FUNCTION_BLOCK MM_TO_PLS
VAR_INPUT
	UINT_PLS_RATIO : UINT;
	UINT_TARGET1_MM : UINT;
	UINT_VEL1_MM : UINT;
	UINT_TARGET2_MM : UINT;
	UINT_VEL2_MM : UINT;
	UINT_TARGET3_MM : UINT;
	UINT_VEL3_MM : UINT;
	UINT_TARGET4_MM : UINT;
	UINT_VEL4_MM : UINT;
	UINT_JOG_2SPD_MM : UINT;
END_VAR

VAR_OUTPUT
	TARGET1_WR_UINT : UINT;
	VEL1_WR_UINT : UINT;
	TARGET2_WR_UINT : UINT;
	VEL2_WR_UINT : UINT;
	TARGET3_WR_UINT : UINT;
	VEL3_WR_UINT : UINT;
	TARGET4_WR_UINT : UINT;
	VEL4_WR_UINT : UINT;
	JOG_2SPD_UINT : UINT;

END_VAR

VAR
END_VAR

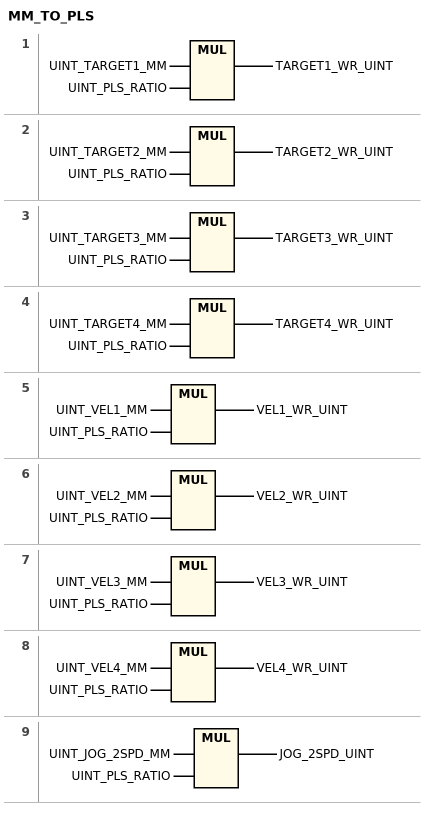
// NETWORK 1
TARGET1_WR_UINT := UINT_TARGET1_MM * UINT_PLS_RATIO;

// NETWORK 2
TARGET2_WR_UINT := UINT_TARGET2_MM * UINT_PLS_RATIO;

// NETWORK 3
TARGET3_WR_UINT := UINT_TARGET3_MM * UINT_PLS_RATIO;

// NETWORK 4
TARGET4_WR_UINT := UINT_TARGET4_MM * UINT_PLS_RATIO;

// NETWORK 5
VEL1_WR_UINT := UINT_VEL1_MM * UINT_PLS_RATIO;

// NETWORK 6
VEL2_WR_UINT := UINT_VEL2_MM * UINT_PLS_RATIO;

// NETWORK 7
VEL3_WR_UINT := UINT_VEL3_MM * UINT_PLS_RATIO;

// NETWORK 8
VEL4_WR_UINT := UINT_VEL4_MM * UINT_PLS_RATIO;

// NETWORK 9
JOG_2SPD_UINT := UINT_JOG_2SPD_MM * UINT_PLS_RATIO;

END_FUNCTION_BLOCK

(* stored: Version 1.1.0.1, ProductVersion 3.1.4024.12
   POU MM_TO_PLS: Id {dbd88c80-a76a-458b-8087-18ab5ca5de8f}, SpecialFunc None *)
